// Mitsubishi GX Works2 project: Main   PLC: FX3U/FX3UC

PROGRAM MAIN
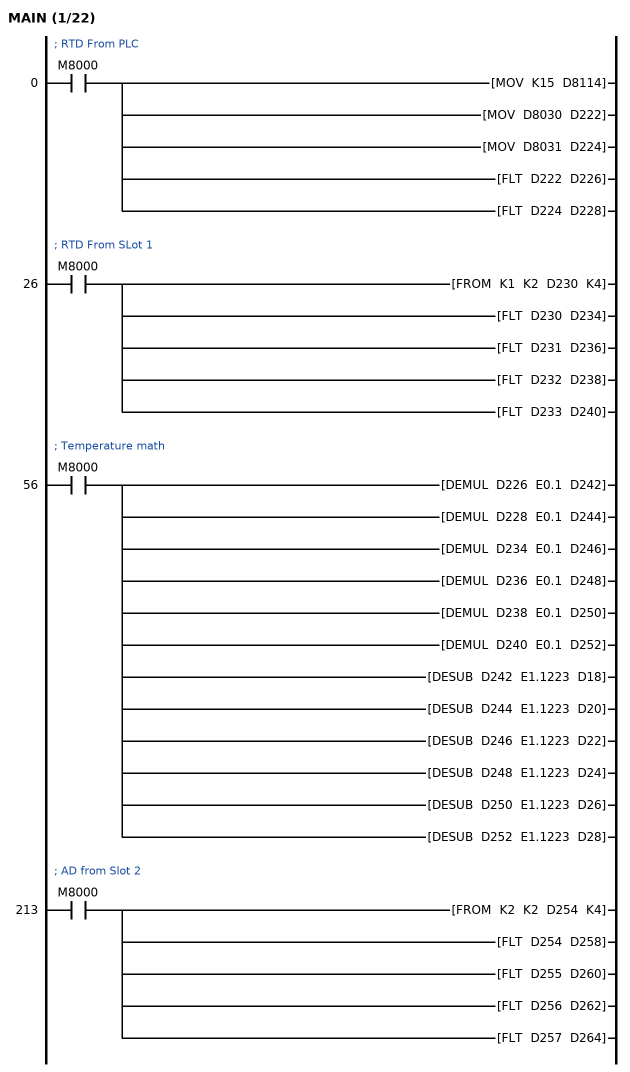
; RTD From PLC
0     LD      M8000
      MOV     K15 D8114
      MOV     D8030 D222
      MOV     D8031 D224
      FLT     D222 D226
      FLT     D224 D228
; RTD From SLot 1
26    LD      M8000
      FROM    K1 K2 D230 K4
      FLT     D230 D234
      FLT     D231 D236
      FLT     D232 D238
      FLT     D233 D240
; Temperature math
56    LD      M8000
      DEMUL   D226 E0.1 D242
      DEMUL   D228 E0.1 D244
      DEMUL   D234 E0.1 D246
      DEMUL   D236 E0.1 D248
      DEMUL   D238 E0.1 D250
      DEMUL   D240 E0.1 D252
      DESUB   D242 E1.1223 D18
      DESUB   D244 E1.1223 D20
      DESUB   D246 E1.1223 D22
      DESUB   D248 E1.1223 D24
      DESUB   D250 E1.1223 D26
      DESUB   D252 E1.1223 D28
; AD from Slot 2
213   LD      M8000
      FROM    K2 K2 D254 K4
      FLT     D254 D258
      FLT     D255 D260
      FLT     D256 D262
      FLT     D257 D264
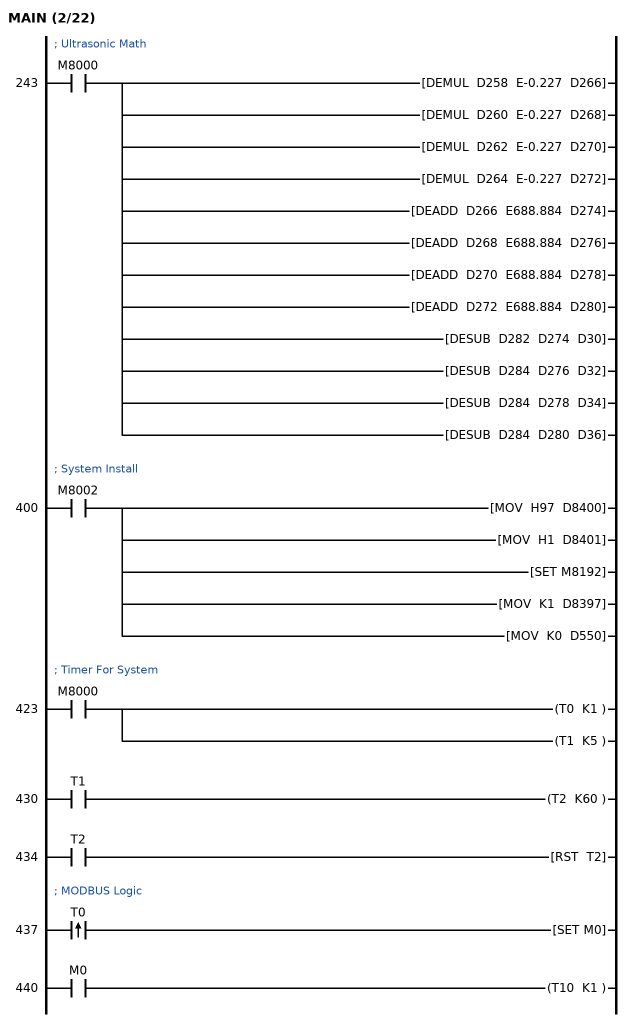
; Ultrasonic Math
243   LD      M8000
      DEMUL   D258 E-0.227 D266
      DEMUL   D260 E-0.227 D268
      DEMUL   D262 E-0.227 D270
      DEMUL   D264 E-0.227 D272
      DEADD   D266 E688.884 D274
      DEADD   D268 E688.884 D276
      DEADD   D270 E688.884 D278
      DEADD   D272 E688.884 D280
      DESUB   D282 D274 D30
      DESUB   D284 D276 D32
      DESUB   D284 D278 D34
      DESUB   D284 D280 D36
; System Install
400   LD      M8002
      MOV     H97 D8400
      MOV     H1 D8401
      SET     M8192
      MOV     K1 D8397
      MOV     K0 D550
; Timer For System
423   LD      M8000
      OUT     T0 K1
      OUT     T1 K5
430   LD      T1
      OUT     T2 K60
434   LD      T2
      RST     T2
; MODBUS Logic
437   LDP     T0
      SET     M0
440   LD      M0
      OUT     T10 K1
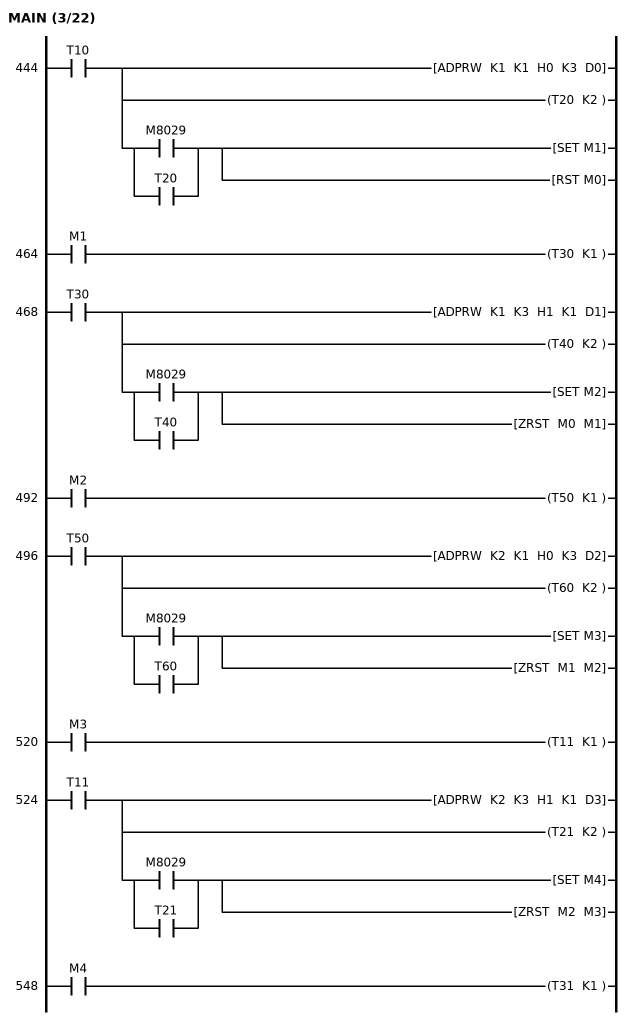
444   LD      T10
      ADPRW   K1 K1 H0 K3 D0
      OUT     T20 K2
      LD      M8029
      OR      T20
      ANB
      SET     M1
      RST     M0
464   LD      M1
      OUT     T30 K1
468   LD      T30
      ADPRW   K1 K3 H1 K1 D1
      OUT     T40 K2
      LD      M8029
      OR      T40
      ANB
      SET     M2
      ZRST    M0 M1
492   LD      M2
      OUT     T50 K1
496   LD      T50
      ADPRW   K2 K1 H0 K3 D2
      OUT     T60 K2
      LD      M8029
      OR      T60
      ANB
      SET     M3
      ZRST    M1 M2
520   LD      M3
      OUT     T11 K1
524   LD      T11
      ADPRW   K2 K3 H1 K1 D3
      OUT     T21 K2
      LD      M8029
      OR      T21
      ANB
      SET     M4
      ZRST    M2 M3
548   LD      M4
      OUT     T31 K1
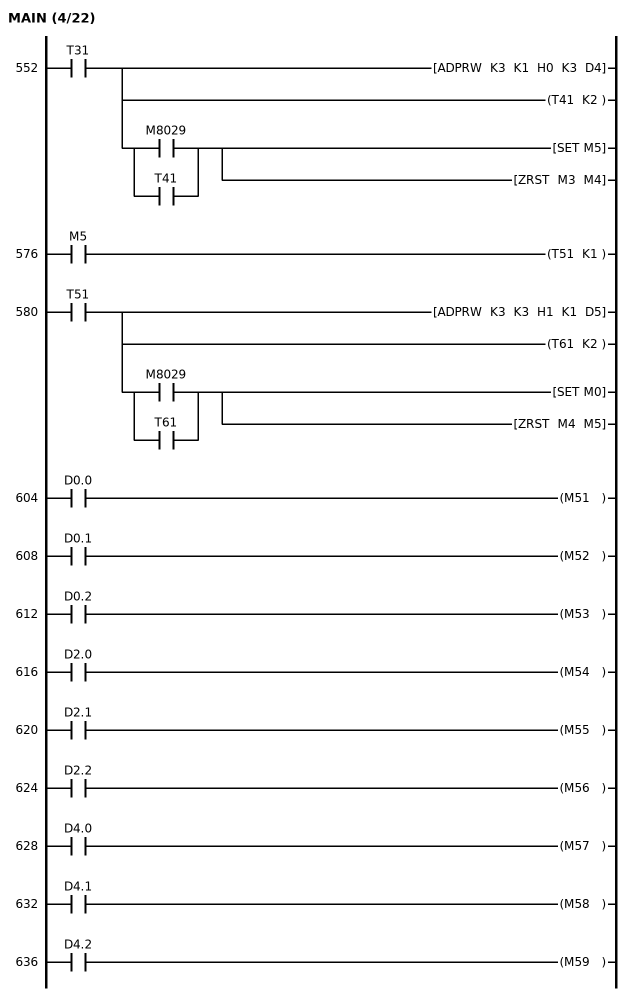
552   LD      T31
      ADPRW   K3 K1 H0 K3 D4
      OUT     T41 K2
      LD      M8029
      OR      T41
      ANB
      SET     M5
      ZRST    M3 M4
576   LD      M5
      OUT     T51 K1
580   LD      T51
      ADPRW   K3 K3 H1 K1 D5
      OUT     T61 K2
      LD      M8029
      OR      T61
      ANB
      SET     M0
      ZRST    M4 M5
604   LD      D0.0
      OUT     M51
608   LD      D0.1
      OUT     M52
612   LD      D0.2
      OUT     M53
616   LD      D2.0
      OUT     M54
620   LD      D2.1
      OUT     M55
624   LD      D2.2
      OUT     M56
628   LD      D4.0
      OUT     M57
632   LD      D4.1
      OUT     M58
636   LD      D4.2
      OUT     M59
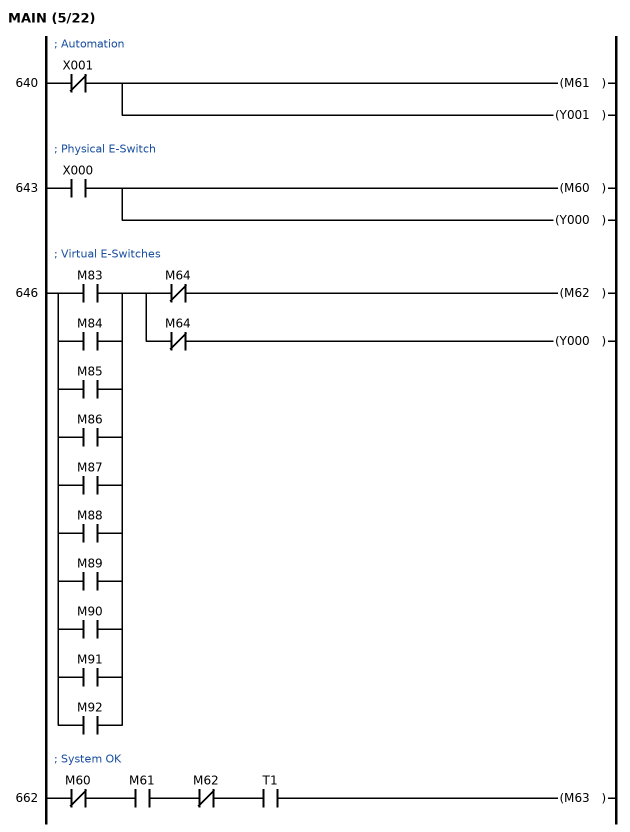
; Automation
640   LDI     X001
      OUT     M61
      OUT     Y001
; Physical E-Switch
643   LD      X000
      OUT     M60
      OUT     Y000
; Virtual E-Switches
646   LD      M83
      OR      M84
      OR      M85
      OR      M86
      OR      M87
      OR      M88
      OR      M89
      OR      M90
      OR      M91
      OR      M92
      MPS
      ANI     M64
      OUT     M62
      MPP
      ANI     M64
      OUT     Y000
; System OK
662   LDI     M60
      AND     M61
      ANI     M62
      AND     T1
      OUT     M63
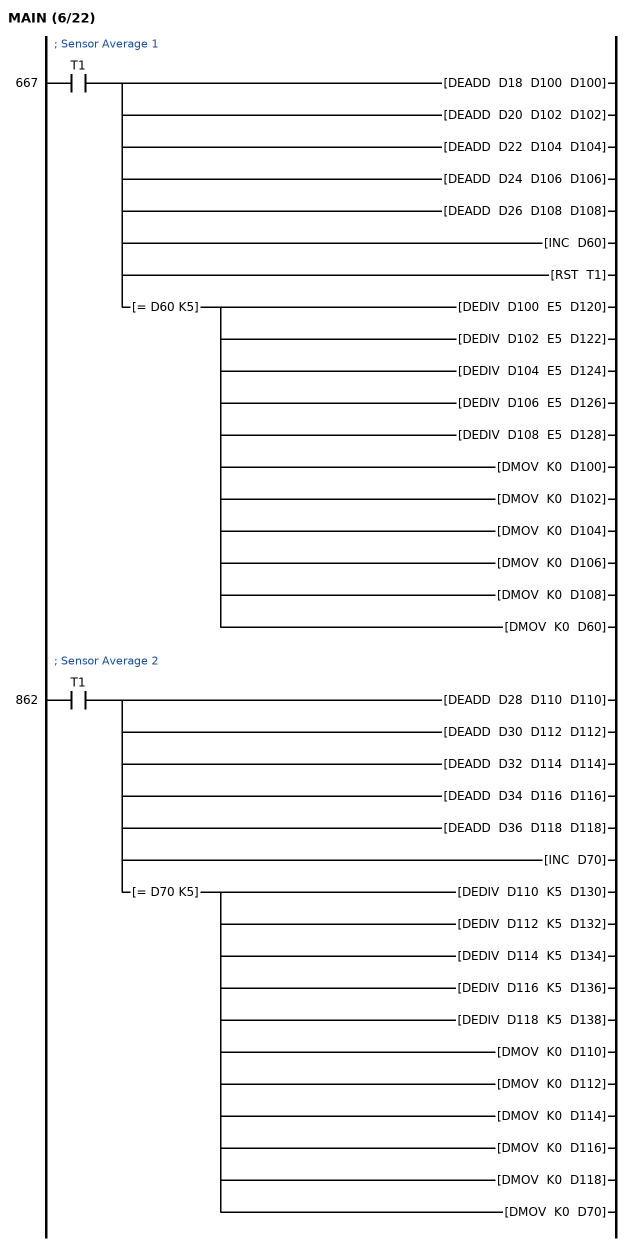
; Sensor Average 1
667   LD      T1
      DEADD   D18 D100 D100
      DEADD   D20 D102 D102
      DEADD   D22 D104 D104
      DEADD   D24 D106 D106
      DEADD   D26 D108 D108
      INC     D60
      RST     T1
      AND=    D60 K5
      DEDIV   D100 E5 D120
      DEDIV   D102 E5 D122
      DEDIV   D104 E5 D124
      DEDIV   D106 E5 D126
      DEDIV   D108 E5 D128
      DMOV    K0 D100
      DMOV    K0 D102
      DMOV    K0 D104
      DMOV    K0 D106
      DMOV    K0 D108
      DMOV    K0 D60
; Sensor Average 2
862   LD      T1
      DEADD   D28 D110 D110
      DEADD   D30 D112 D112
      DEADD   D32 D114 D114
      DEADD   D34 D116 D116
      DEADD   D36 D118 D118
      INC     D70
      AND=    D70 K5
      DEDIV   D110 K5 D130
      DEDIV   D112 K5 D132
      DEDIV   D114 K5 D134
      DEDIV   D116 K5 D136
      DEDIV   D118 K5 D138
      DMOV    K0 D110
      DMOV    K0 D112
      DMOV    K0 D114
      DMOV    K0 D116
      DMOV    K0 D118
      DMOV    K0 D70
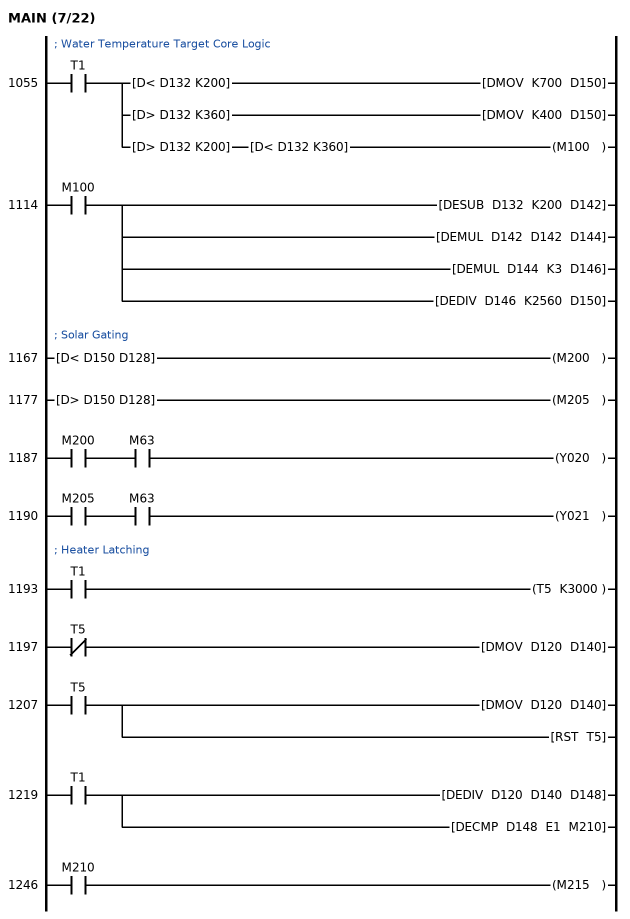
; Water Temperature Target Core Logic
1055  LD      T1
      MPS
      ANDD<   D132 K200
      DMOV    K700 D150
      MRD
      ANDD>   D132 K360
      DMOV    K400 D150
      MPP
      ANDD>   D132 K200
      ANDD<   D132 K360
      OUT     M100
1114  LD      M100
      DESUB   D132 K200 D142
      DEMUL   D142 D142 D144
      DEMUL   D144 K3 D146
      DEDIV   D146 K2560 D150
; Solar Gating
1167  LDD<    D150 D128
      OUT     M200
1177  LDD>    D150 D128
      OUT     M205
1187  LD      M200
      AND     M63
      OUT     Y020
1190  LD      M205
      AND     M63
      OUT     Y021
; Heater Latching
1193  LD      T1
      OUT     T5 K3000
1197  LDI     T5
      DMOV    D120 D140
1207  LD      T5
      DMOV    D120 D140
      RST     T5
1219  LD      T1
      DEDIV   D120 D140 D148
      DECMP   D148 E1 M210
1246  LD      M210
      OUT     M215
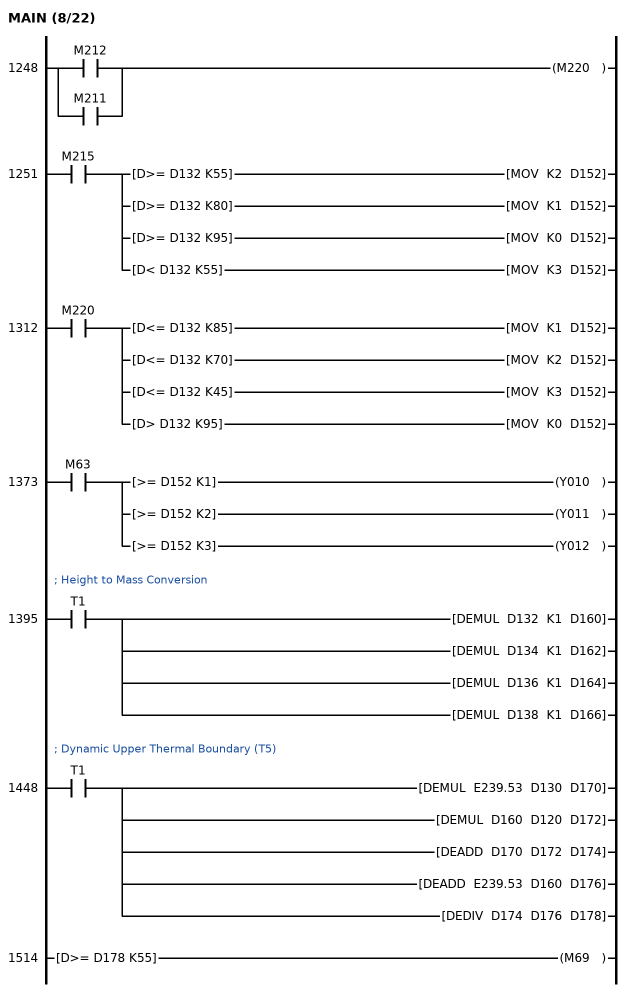
1248  LD      M212
      OR      M211
      OUT     M220
1251  LD      M215
      MPS
      ANDD>=  D132 K55
      MOV     K2 D152
      MRD
      ANDD>=  D132 K80
      MOV     K1 D152
      MRD
      ANDD>=  D132 K95
      MOV     K0 D152
      MPP
      ANDD<   D132 K55
      MOV     K3 D152
1312  LD      M220
      MPS
      ANDD<=  D132 K85
      MOV     K1 D152
      MRD
      ANDD<=  D132 K70
      MOV     K2 D152
      MRD
      ANDD<=  D132 K45
      MOV     K3 D152
      MPP
      ANDD>   D132 K95
      MOV     K0 D152
1373  LD      M63
      MPS
      AND>=   D152 K1
      OUT     Y010
      MRD
      AND>=   D152 K2
      OUT     Y011
      MPP
      AND>=   D152 K3
      OUT     Y012
; Height to Mass Conversion
1395  LD      T1
      DEMUL   D132 K1 D160
      DEMUL   D134 K1 D162
      DEMUL   D136 K1 D164
      DEMUL   D138 K1 D166
; Dynamic Upper Thermal Boundary (T5)
1448  LD      T1
      DEMUL   E239.53 D130 D170
      DEMUL   D160 D120 D172
      DEADD   D170 D172 D174
      DEADD   E239.53 D160 D176
      DEDIV   D174 D176 D178
1514  LDD>=   D178 K55
      OUT     M69
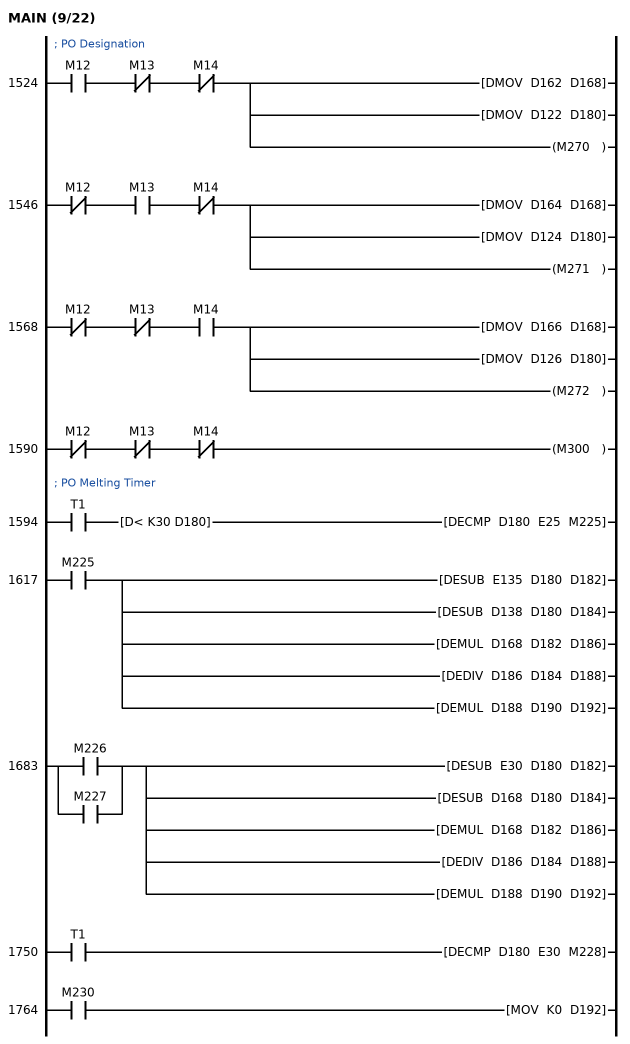
; PO Designation
1524  LD      M12
      ANI     M13
      ANI     M14
      DMOV    D162 D168
      DMOV    D122 D180
      OUT     M270
1546  LDI     M12
      AND     M13
      ANI     M14
      DMOV    D164 D168
      DMOV    D124 D180
      OUT     M271
1568  LDI     M12
      ANI     M13
      AND     M14
      DMOV    D166 D168
      DMOV    D126 D180
      OUT     M272
1590  LDI     M12
      ANI     M13
      ANI     M14
      OUT     M300
; PO Melting Timer
1594  LD      T1
      ANDD<   K30 D180
      DECMP   D180 E25 M225
1617  LD      M225
      DESUB   E135 D180 D182
      DESUB   D138 D180 D184
      DEMUL   D168 D182 D186
      DEDIV   D186 D184 D188
      DEMUL   D188 D190 D192
1683  LD      M226
      OR      M227
      DESUB   E30 D180 D182
      DESUB   D168 D180 D184
      DEMUL   D168 D182 D186
      DEDIV   D186 D184 D188
      DEMUL   D188 D190 D192
1750  LD      T1
      DECMP   D180 E30 M228
1764  LD      M230
      MOV     K0 D192
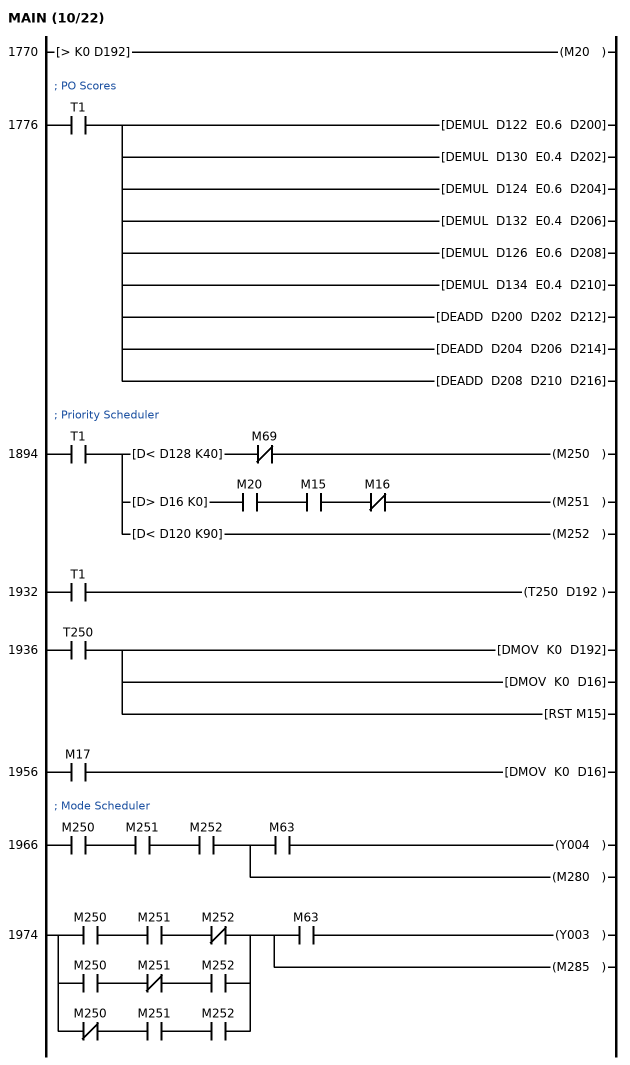
1770  LD>     K0 D192
      OUT     M20
; PO Scores
1776  LD      T1
      DEMUL   D122 E0.6 D200
      DEMUL   D130 E0.4 D202
      DEMUL   D124 E0.6 D204
      DEMUL   D132 E0.4 D206
      DEMUL   D126 E0.6 D208
      DEMUL   D134 E0.4 D210
      DEADD   D200 D202 D212
      DEADD   D204 D206 D214
      DEADD   D208 D210 D216
; Priority Scheduler
1894  LD      T1
      MPS
      ANDD<   D128 K40
      ANI     M69
      OUT     M250
      MRD
      ANDD>   D16 K0
      AND     M20
      AND     M15
      ANI     M16
      OUT     M251
      MPP
      ANDD<   D120 K90
      OUT     M252
1932  LD      T1
      OUT     T250 D192
1936  LD      T250
      DMOV    K0 D192
      DMOV    K0 D16
      RST     M15
1956  LD      M17
      DMOV    K0 D16
; Mode Scheduler
1966  LD      M250
      AND     M251
      AND     M252
      MPS
      AND     M63
      OUT     Y004
      MPP
      OUT     M280
1974  LD      M250
      AND     M251
      ANI     M252
      LD      M250
      ANI     M251
      AND     M252
      ORB
      LDI     M250
      AND     M251
      AND     M252
      ORB
      MPS
      AND     M63
      OUT     Y003
      MPP
      OUT     M285
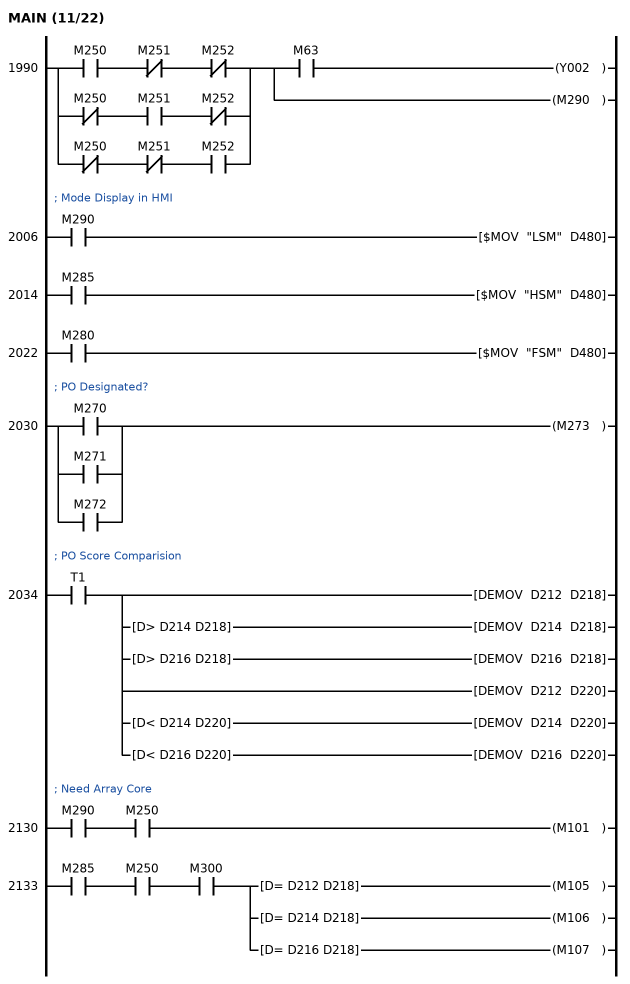
1990  LD      M250
      ANI     M251
      ANI     M252
      LDI     M250
      AND     M251
      ANI     M252
      ORB
      LDI     M250
      ANI     M251
      AND     M252
      ORB
      MPS
      AND     M63
      OUT     Y002
      MPP
      OUT     M290
; Mode Display in HMI
2006  LD      M290
      $MOV    "LSM" D480
2014  LD      M285
      $MOV    "HSM" D480
2022  LD      M280
      $MOV    "FSM" D480
; PO Designated?
2030  LD      M270
      OR      M271
      OR      M272
      OUT     M273
; PO Score Comparision
2034  LD      T1
      DEMOV   D212 D218
      MPS
      ANDD>   D214 D218
      DEMOV   D214 D218
      MRD
      ANDD>   D216 D218
      DEMOV   D216 D218
      MPP
      DEMOV   D212 D220
      MPS
      ANDD<   D214 D220
      DEMOV   D214 D220
      MPP
      ANDD<   D216 D220
      DEMOV   D216 D220
; Need Array Core
2130  LD      M290
      AND     M250
      OUT     M101
2133  LD      M285
      AND     M250
      AND     M300
      MPS
      ANDD=   D212 D218
      OUT     M105
      MRD
      ANDD=   D214 D218
      OUT     M106
      MPP
      ANDD=   D216 D218
      OUT     M107
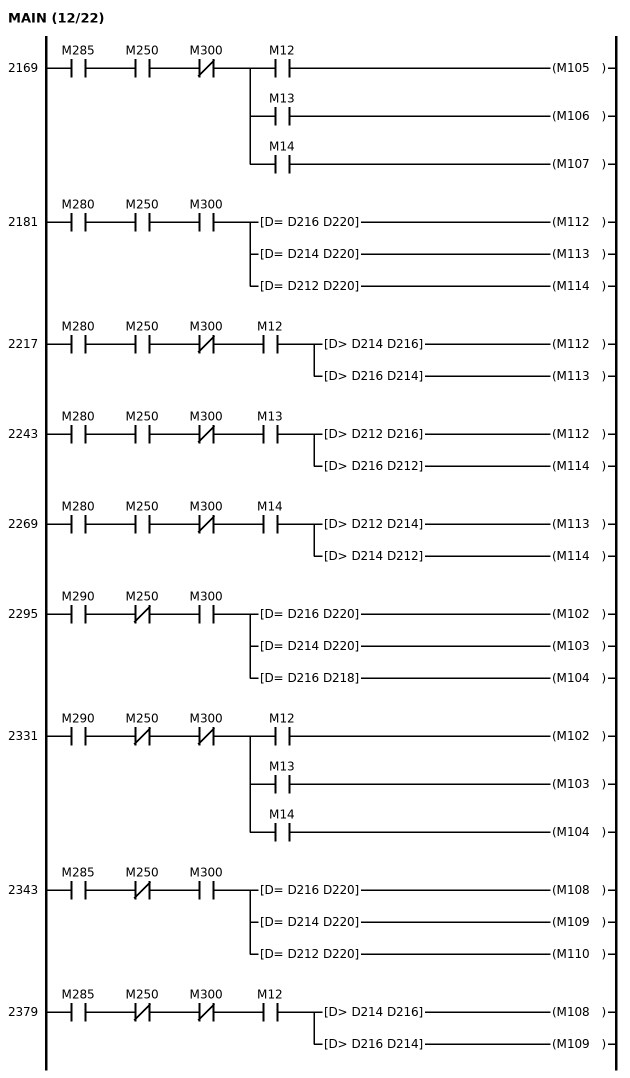
2169  LD      M285
      AND     M250
      ANI     M300
      MPS
      AND     M12
      OUT     M105
      MRD
      AND     M13
      OUT     M106
      MPP
      AND     M14
      OUT     M107
2181  LD      M280
      AND     M250
      AND     M300
      MPS
      ANDD=   D216 D220
      OUT     M112
      MRD
      ANDD=   D214 D220
      OUT     M113
      MPP
      ANDD=   D212 D220
      OUT     M114
2217  LD      M280
      AND     M250
      ANI     M300
      AND     M12
      MPS
      ANDD>   D214 D216
      OUT     M112
      MPP
      ANDD>   D216 D214
      OUT     M113
2243  LD      M280
      AND     M250
      ANI     M300
      AND     M13
      MPS
      ANDD>   D212 D216
      OUT     M112
      MPP
      ANDD>   D216 D212
      OUT     M114
2269  LD      M280
      AND     M250
      ANI     M300
      AND     M14
      MPS
      ANDD>   D212 D214
      OUT     M113
      MPP
      ANDD>   D214 D212
      OUT     M114
2295  LD      M290
      ANI     M250
      AND     M300
      MPS
      ANDD=   D216 D220
      OUT     M102
      MRD
      ANDD=   D214 D220
      OUT     M103
      MPP
      ANDD=   D216 D218
      OUT     M104
2331  LD      M290
      ANI     M250
      ANI     M300
      MPS
      AND     M12
      OUT     M102
      MRD
      AND     M13
      OUT     M103
      MPP
      AND     M14
      OUT     M104
2343  LD      M285
      ANI     M250
      AND     M300
      MPS
      ANDD=   D216 D220
      OUT     M108
      MRD
      ANDD=   D214 D220
      OUT     M109
      MPP
      ANDD=   D212 D220
      OUT     M110
2379  LD      M285
      ANI     M250
      ANI     M300
      AND     M12
      MPS
      ANDD>   D214 D216
      OUT     M108
      MPP
      ANDD>   D216 D214
      OUT     M109
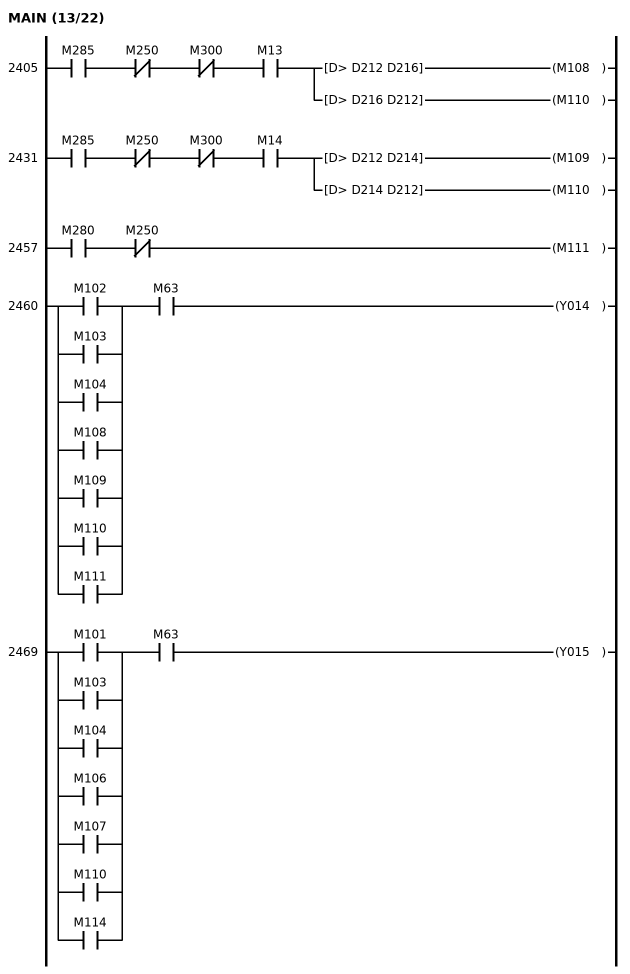
2405  LD      M285
      ANI     M250
      ANI     M300
      AND     M13
      MPS
      ANDD>   D212 D216
      OUT     M108
      MPP
      ANDD>   D216 D212
      OUT     M110
2431  LD      M285
      ANI     M250
      ANI     M300
      AND     M14
      MPS
      ANDD>   D212 D214
      OUT     M109
      MPP
      ANDD>   D214 D212
      OUT     M110
2457  LD      M280
      ANI     M250
      OUT     M111
2460  LD      M102
      OR      M103
      OR      M104
      OR      M108
      OR      M109
      OR      M110
      OR      M111
      AND     M63
      OUT     Y014
2469  LD      M101
      OR      M103
      OR      M104
      OR      M106
      OR      M107
      OR      M110
      OR      M114
      AND     M63
      OUT     Y015
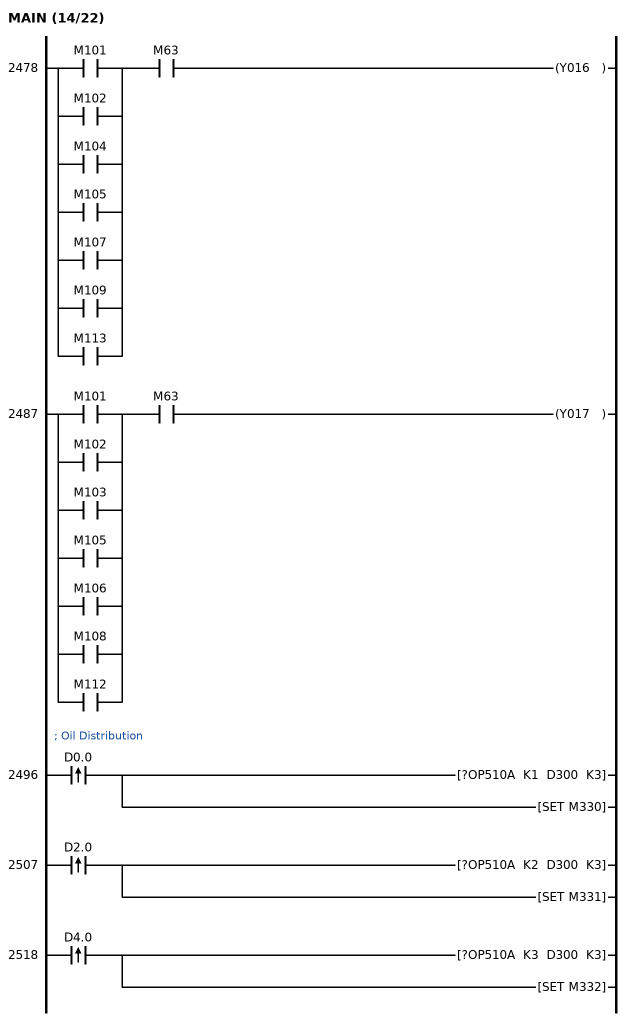
2478  LD      M101
      OR      M102
      OR      M104
      OR      M105
      OR      M107
      OR      M109
      OR      M113
      AND     M63
      OUT     Y016
2487  LD      M101
      OR      M102
      OR      M103
      OR      M105
      OR      M106
      OR      M108
      OR      M112
      AND     M63
      OUT     Y017
; Oil Distribution
2496  LDP     D0.0
      ?OP510A K1 D300 K3
      SET     M330
2507  LDP     D2.0
      ?OP510A K2 D300 K3
      SET     M331
2518  LDP     D4.0
      ?OP510A K3 D300 K3
      SET     M332
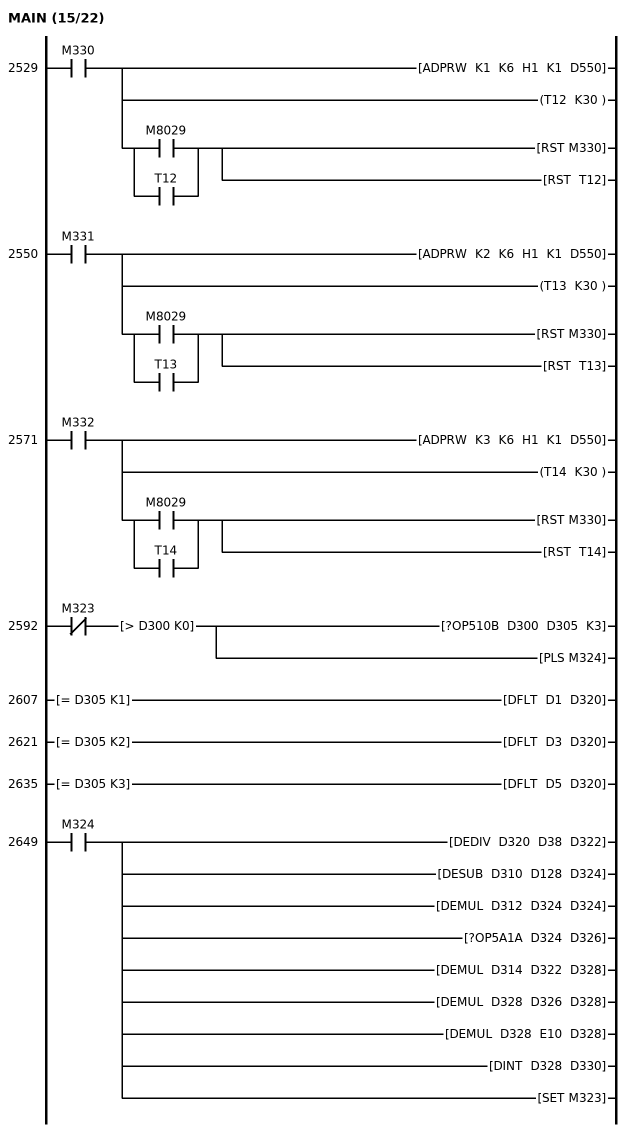
2529  LD      M330
      ADPRW   K1 K6 H1 K1 D550
      OUT     T12 K30
      LD      M8029
      OR      T12
      ANB
      RST     M330
      RST     T12
2550  LD      M331
      ADPRW   K2 K6 H1 K1 D550
      OUT     T13 K30
      LD      M8029
      OR      T13
      ANB
      RST     M330
      RST     T13
2571  LD      M332
      ADPRW   K3 K6 H1 K1 D550
      OUT     T14 K30
      LD      M8029
      OR      T14
      ANB
      RST     M330
      RST     T14
2592  LDI     M323
      AND>    D300 K0
      ?OP510B D300 D305 K3
      PLS     M324
2607  LD=     D305 K1
      DFLT    D1 D320
2621  LD=     D305 K2
      DFLT    D3 D320
2635  LD=     D305 K3
      DFLT    D5 D320
2649  LD      M324
      DEDIV   D320 D38 D322
      DESUB   D310 D128 D324
      DEMUL   D312 D324 D324
      ?OP5A1A D324 D326
      DEMUL   D314 D322 D328
      DEMUL   D328 D326 D328
      DEMUL   D328 E10 D328
      DINT    D328 D330
      SET     M323
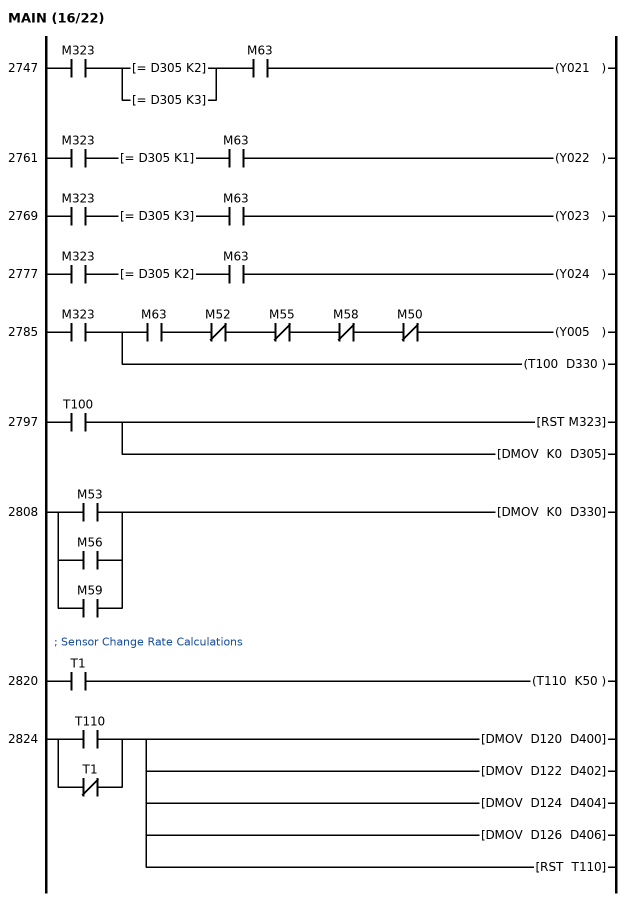
2747  LD      M323
      LD=     D305 K2
      OR=     D305 K3
      ANB
      AND     M63
      OUT     Y021
2761  LD      M323
      AND=    D305 K1
      AND     M63
      OUT     Y022
2769  LD      M323
      AND=    D305 K3
      AND     M63
      OUT     Y023
2777  LD      M323
      AND=    D305 K2
      AND     M63
      OUT     Y024
2785  LD      M323
      MPS
      AND     M63
      ANI     M52
      ANI     M55
      ANI     M58
      ANI     M50
      OUT     Y005
      MPP
      OUT     T100 D330
2797  LD      T100
      RST     M323
      DMOV    K0 D305
2808  LD      M53
      OR      M56
      OR      M59
      DMOV    K0 D330
; Sensor Change Rate Calculations
2820  LD      T1
      OUT     T110 K50
2824  LD      T110
      ORI     T1
      DMOV    D120 D400
      DMOV    D122 D402
      DMOV    D124 D404
      DMOV    D126 D406
      RST     T110
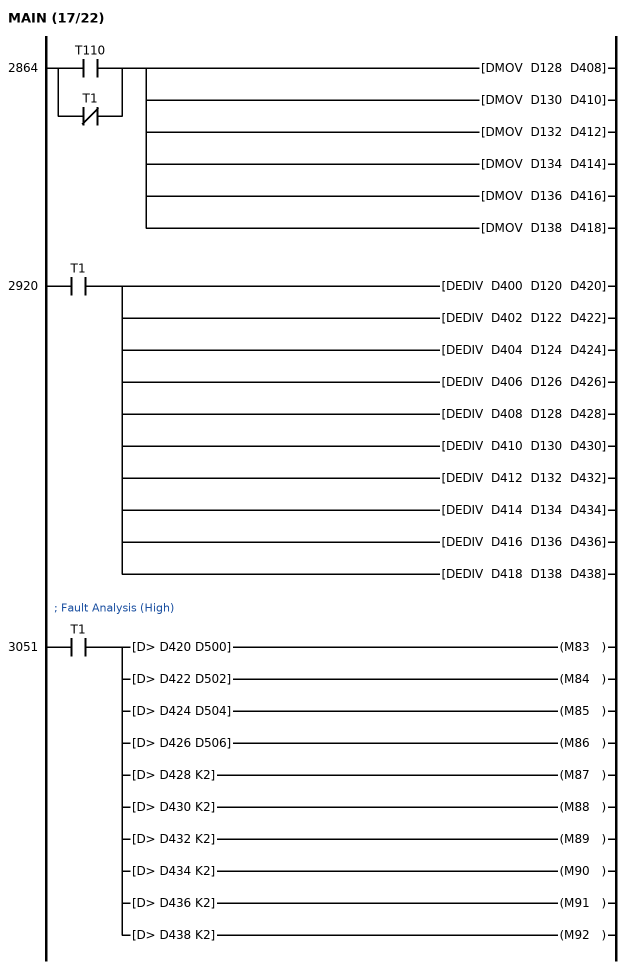
2864  LD      T110
      ORI     T1
      DMOV    D128 D408
      DMOV    D130 D410
      DMOV    D132 D412
      DMOV    D134 D414
      DMOV    D136 D416
      DMOV    D138 D418
2920  LD      T1
      DEDIV   D400 D120 D420
      DEDIV   D402 D122 D422
      DEDIV   D404 D124 D424
      DEDIV   D406 D126 D426
      DEDIV   D408 D128 D428
      DEDIV   D410 D130 D430
      DEDIV   D412 D132 D432
      DEDIV   D414 D134 D434
      DEDIV   D416 D136 D436
      DEDIV   D418 D138 D438
; Fault Analysis (High)
3051  LD      T1
      MPS
      ANDD>   D420 D500
      OUT     M83
      MRD
      ANDD>   D422 D502
      OUT     M84
      MRD
      ANDD>   D424 D504
      OUT     M85
      MRD
      ANDD>   D426 D506
      OUT     M86
      MRD
      ANDD>   D428 K2
      OUT     M87
      MRD
      ANDD>   D430 K2
      OUT     M88
      MRD
      ANDD>   D432 K2
      OUT     M89
      MRD
      ANDD>   D434 K2
      OUT     M90
      MRD
      ANDD>   D436 K2
      OUT     M91
      MPP
      ANDD>   D438 K2
      OUT     M92
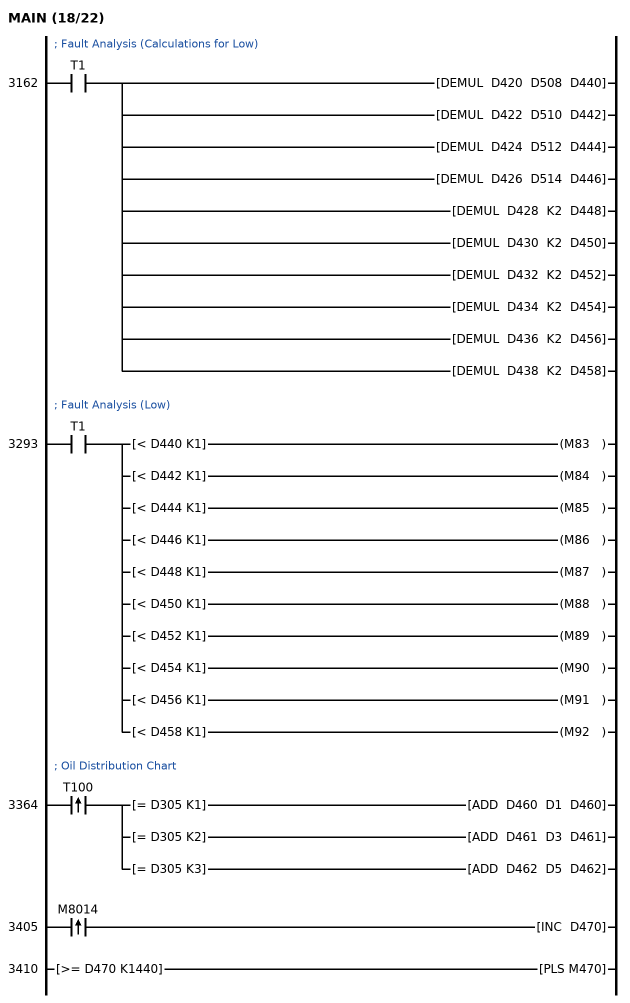
; Fault Analysis (Calculations for Low)
3162  LD      T1
      DEMUL   D420 D508 D440
      DEMUL   D422 D510 D442
      DEMUL   D424 D512 D444
      DEMUL   D426 D514 D446
      DEMUL   D428 K2 D448
      DEMUL   D430 K2 D450
      DEMUL   D432 K2 D452
      DEMUL   D434 K2 D454
      DEMUL   D436 K2 D456
      DEMUL   D438 K2 D458
; Fault Analysis (Low)
3293  LD      T1
      MPS
      AND<    D440 K1
      OUT     M83
      MRD
      AND<    D442 K1
      OUT     M84
      MRD
      AND<    D444 K1
      OUT     M85
      MRD
      AND<    D446 K1
      OUT     M86
      MRD
      AND<    D448 K1
      OUT     M87
      MRD
      AND<    D450 K1
      OUT     M88
      MRD
      AND<    D452 K1
      OUT     M89
      MRD
      AND<    D454 K1
      OUT     M90
      MRD
      AND<    D456 K1
      OUT     M91
      MPP
      AND<    D458 K1
      OUT     M92
; Oil Distribution Chart
3364  LDP     T100
      MPS
      AND=    D305 K1
      ADD     D460 D1 D460
      MRD
      AND=    D305 K2
      ADD     D461 D3 D461
      MPP
      AND=    D305 K3
      ADD     D462 D5 D462
3405  LDP     M8014
      INC     D470
3410  LD>=    D470 K1440
      PLS     M470
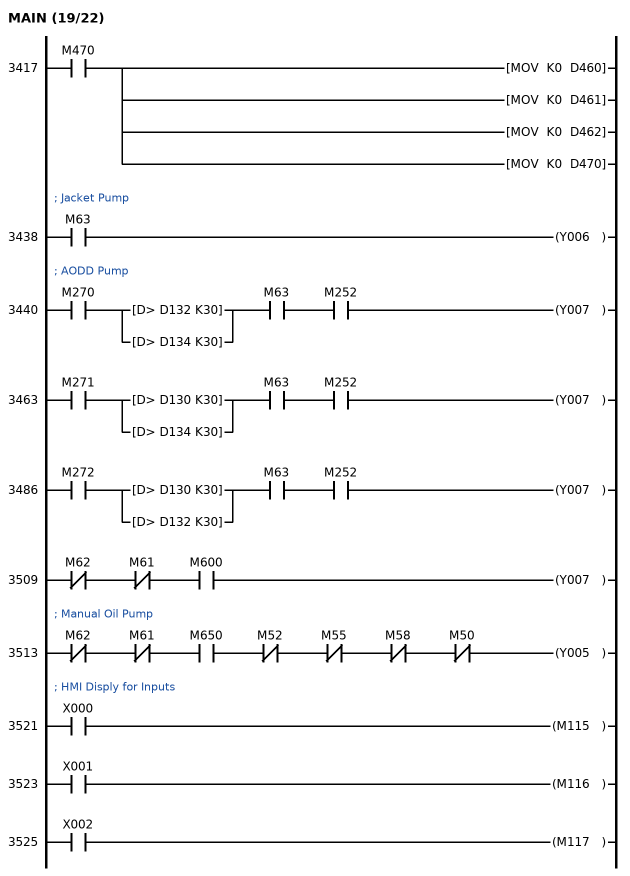
3417  LD      M470
      MOV     K0 D460
      MOV     K0 D461
      MOV     K0 D462
      MOV     K0 D470
; Jacket Pump
3438  LD      M63
      OUT     Y006
; AODD Pump
3440  LD      M270
      LDD>    D132 K30
      ORD>    D134 K30
      ANB
      AND     M63
      AND     M252
      OUT     Y007
3463  LD      M271
      LDD>    D130 K30
      ORD>    D134 K30
      ANB
      AND     M63
      AND     M252
      OUT     Y007
3486  LD      M272
      LDD>    D130 K30
      ORD>    D132 K30
      ANB
      AND     M63
      AND     M252
      OUT     Y007
3509  LDI     M62
      ANI     M61
      AND     M600
      OUT     Y007
; Manual Oil Pump
3513  LDI     M62
      ANI     M61
      AND     M650
      ANI     M52
      ANI     M55
      ANI     M58
      ANI     M50
      OUT     Y005
; HMI Disply for Inputs
3521  LD      X000
      OUT     M115
3523  LD      X001
      OUT     M116
3525  LD      X002
      OUT     M117
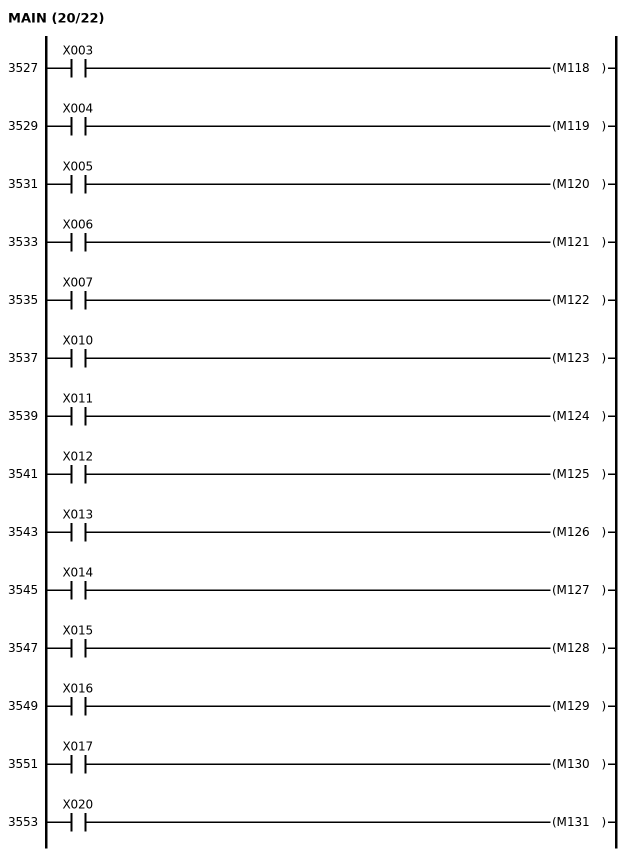
3527  LD      X003
      OUT     M118
3529  LD      X004
      OUT     M119
3531  LD      X005
      OUT     M120
3533  LD      X006
      OUT     M121
3535  LD      X007
      OUT     M122
3537  LD      X010
      OUT     M123
3539  LD      X011
      OUT     M124
3541  LD      X012
      OUT     M125
3543  LD      X013
      OUT     M126
3545  LD      X014
      OUT     M127
3547  LD      X015
      OUT     M128
3549  LD      X016
      OUT     M129
3551  LD      X017
      OUT     M130
3553  LD      X020
      OUT     M131
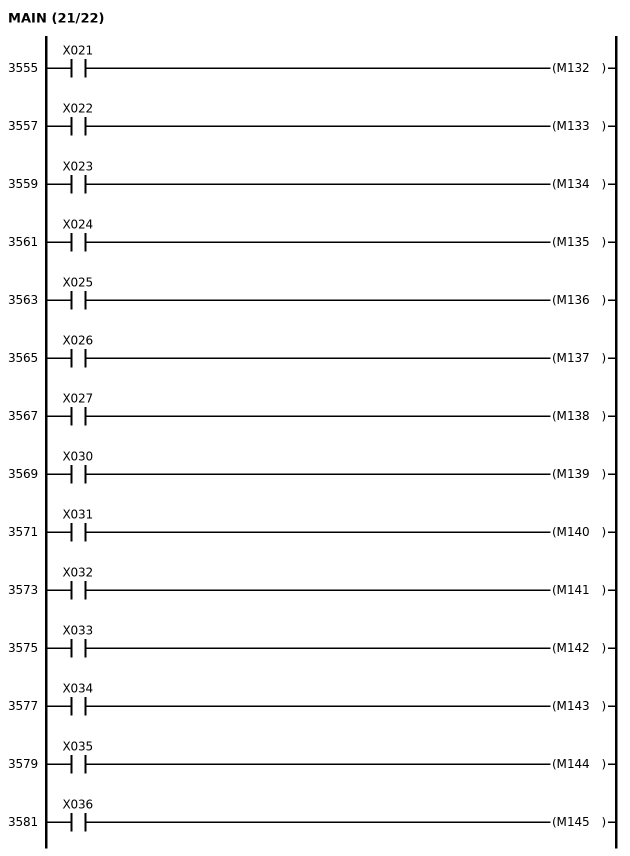
3555  LD      X021
      OUT     M132
3557  LD      X022
      OUT     M133
3559  LD      X023
      OUT     M134
3561  LD      X024
      OUT     M135
3563  LD      X025
      OUT     M136
3565  LD      X026
      OUT     M137
3567  LD      X027
      OUT     M138
3569  LD      X030
      OUT     M139
3571  LD      X031
      OUT     M140
3573  LD      X032
      OUT     M141
3575  LD      X033
      OUT     M142
3577  LD      X034
      OUT     M143
3579  LD      X035
      OUT     M144
3581  LD      X036
      OUT     M145
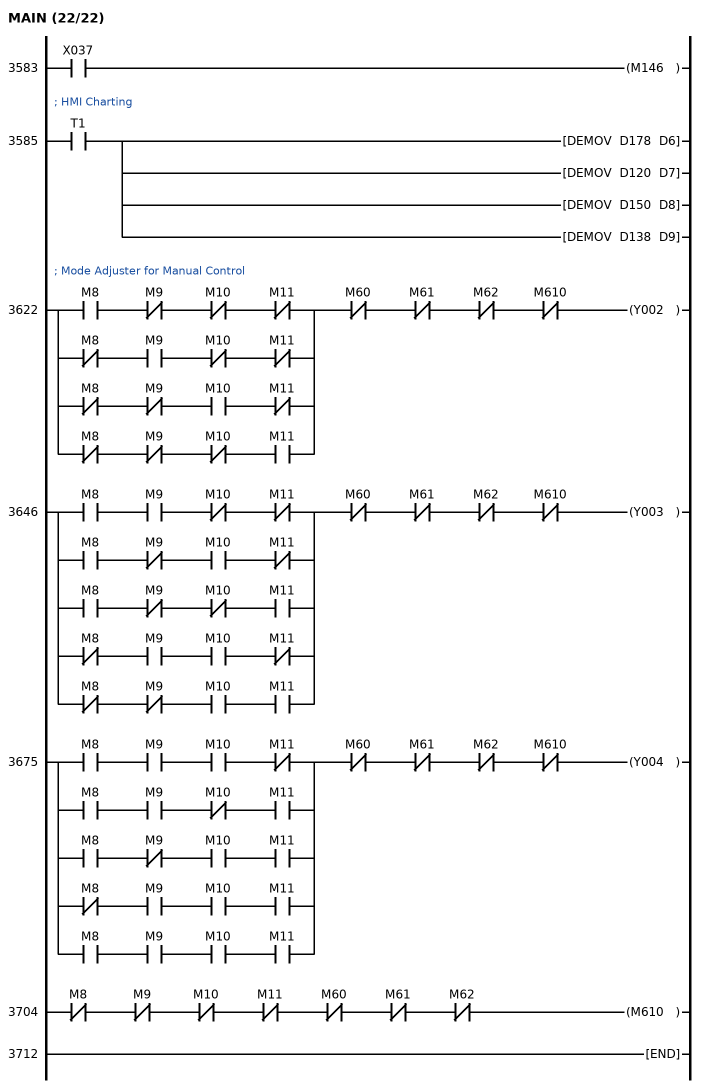
3583  LD      X037
      OUT     M146
; HMI Charting
3585  LD      T1
      DEMOV   D178 D6
      DEMOV   D120 D7
      DEMOV   D150 D8
      DEMOV   D138 D9
; Mode Adjuster for Manual Control
3622  LD      M8
      ANI     M9
      ANI     M10
      ANI     M11
      LDI     M8
      AND     M9
      ANI     M10
      ANI     M11
      ORB
      LDI     M8
      ANI     M9
      AND     M10
      ANI     M11
      ORB
      LDI     M8
      ANI     M9
      ANI     M10
      AND     M11
      ORB
      ANI     M60
      ANI     M61
      ANI     M62
      ANI     M610
      OUT     Y002
3646  LD      M8
      AND     M9
      ANI     M10
      ANI     M11
      LD      M8
      ANI     M9
      AND     M10
      ANI     M11
      ORB
      LD      M8
      ANI     M9
      ANI     M10
      AND     M11
      ORB
      LDI     M8
      AND     M9
      AND     M10
      ANI     M11
      ORB
      LDI     M8
      ANI     M9
      AND     M10
      AND     M11
      ORB
      ANI     M60
      ANI     M61
      ANI     M62
      ANI     M610
      OUT     Y003
3675  LD      M8
      AND     M9
      AND     M10
      ANI     M11
      LD      M8
      AND     M9
      ANI     M10
      AND     M11
      ORB
      LD      M8
      ANI     M9
      AND     M10
      AND     M11
      ORB
      LDI     M8
      AND     M9
      AND     M10
      AND     M11
      ORB
      LD      M8
      AND     M9
      AND     M10
      AND     M11
      ORB
      ANI     M60
      ANI     M61
      ANI     M62
      ANI     M610
      OUT     Y004
3704  LDI     M8
      ANI     M9
      ANI     M10
      ANI     M11
      ANI     M60
      ANI     M61
      ANI     M62
      OUT     M610
3712  END
END_PROGRAM
